FUNCTION togglePvBoost : BOOL
VAR_INPUT
	pMachine : POINTER TO FB_StateMachine;
END_VAR
VAR
END_VAR

IF pMachine^.pd.sensor.photovoltaicBoost = FALSE THEN
	LogMessage(E_LogType.INFO, 'PV Boost wurde geklickt: -> ', 'Ein');	
	pMachine^.pd.sensor.photovoltaicBoost := TRUE;
ELSE
	LogMessage(E_LogType.INFO, 'PV Boost wurde geklickt: -> ', 'Aus');	
	pMachine^.pd.sensor.photovoltaicBoost := FALSE;
END_IF

END_FUNCTION

(* stored: Version 1.1.0.1
   POU togglePvBoost: Id {c034a06b-5db7-4075-99b0-b658a8d8fbee}, SpecialFunc None *)
